PROGRAM Machine_Status
VAR
	AirKnife_Status_String : STRING;
	AirKnife_Disconnected : BOOL;
	AirKnife_Connected : bool;
	
	Rotor_Status_String : STRING;
	Rotor_Disconnected : BOOL;
	
	Feedroll_Status_String : STRING;
	Feedroll_Disconnected : BOOL;
	
	Pelletizer_Status_String : STRING;
	
	Waterbath_Status_String : STRING;
	Waterbath_Disconnected : BOOL;
	Waterbath_Connected : BOOL;
	
END_VAR


Rotor_Status_String := SlaveStatus_FB(GVL_Pelletizer.MyPelletizer.Rotor_VFD.VFD_Connection_Status, Slave_Disconnected => Rotor_Disconnected);
Feedroll_Status_String := SlaveStatus_FB(GVL_Pelletizer.MyPelletizer.Feedroll_VFD.VFD_Connection_Status, Slave_Disconnected => Feedroll_Disconnected);

IF Rotor_Disconnected OR Feedroll_Disconnected THEN
	Pelletizer_Status_String := CONCAT(Rotor_Status_String, Feedroll_Status_String);
ELSE
	Pelletizer_Status_String := 'Slave in OP state';
END_IF


AirKnife_Status_String := SlaveStatus_FB(GVL_AirKnife.AirKnife_VFD.VFD_Connection_Status, Slave_Disconnected => AirKnife_Disconnected);
AirKnife_connected := NOT Airknife_Disconnected;

Waterbath_Status_String := SlaveStatus_FB(GVL_Waterbath.Waterbath_Connection_Status, Slave_Disconnected => Waterbath_Disconnected);
Waterbath_Connected := NOT Waterbath_Disconnected;

END_PROGRAM

(* stored: Version 1.1.0.1, ProductVersion 3.1.4026.11
   POU Machine_Status: Id {0fb206cd-a8a2-4a59-bc2b-cd719b567cca}, SpecialFunc None *)
